ABB RobotStudio station: PickPlace_Station.rspag

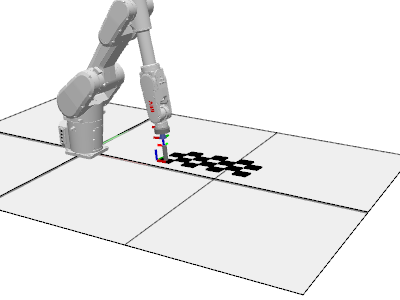
--- station ---
Station PickPlace_Station (saved by RobotStudio 24.3.10835.0)
Controller Controller1
  mechanical unit ROB_1: IRB1300F_7_140__01, 6 joints, base frame (0, 0, 0) mm
Layout (positions relative to the parent item):
  - IRB1300F_7_140__01 [mechanism, from %ABB.RobotStudio.Models.IRB1300%\IRB1300F_7_140__01.rslib] at (0, 0, 0) mm; joint values [-0.071, 0.5331, 0.806, 0.0627, 0.1234, -0.1329] (rad or m)
  - Vacuum 1x1 [part, from User Files\Vacuum 1x1.rslib] at (644.53, -45.15, 299.98) mm, rotated rx -180 ry 6.24 rz 180 deg
  - BlackSquare [part], size 100 x 60 x 10 mm
  - ChessBoard [graphiccomponentgroup] at (-2.34, 163.38, 0) mm, rotated rx 1.02 ry -6.15 rz -9.46 deg
    - MatrixRepeater [smart component, from Components\MatrixRepeater.rslib] at (653.18, -125.32, 0) mm
        properties: Source=BlackSquare; CountX=4; CountY=2; CountZ=1; OffsetX=0.2; OffsetY=0.12; OffsetZ=0.1
      - Objet_1 [part], size 100 x 60 x 10 mm
      - Objet_1 [part] at (200, 0, 0) mm, size 100 x 60 x 10 mm
      - Objet_1 [part] at (400, 0, 0) mm, size 100 x 60 x 10 mm
      - Objet_1 [part] at (600, 0, 0) mm, size 100 x 60 x 10 mm
      - Objet_1 [part] at (0, 120, 0) mm, size 100 x 60 x 10 mm
      - Objet_1 [part] at (200, 120, 0) mm, size 100 x 60 x 10 mm
      - Objet_1 [part] at (400, 120, 0) mm, size 100 x 60 x 10 mm
      - Objet_1 [part] at (600, 120, 0) mm, size 100 x 60 x 10 mm
    - MatrixRepeater_2 [smart component, from Components\MatrixRepeater.rslib] at (751.9, -66.74, 0) mm
        properties: Source=BlackSquare; CountX=3; CountY=2; CountZ=1; OffsetX=0.2; OffsetY=0.12; OffsetZ=0.1
      - Objet_1 [part], size 100 x 60 x 10 mm
      - Objet_1 [part] at (200, 0, 0) mm, size 100 x 60 x 10 mm
      - Objet_1 [part] at (400, 0, 0) mm, size 100 x 60 x 10 mm
      - Objet_1 [part] at (0, 120, 0) mm, size 100 x 60 x 10 mm
      - Objet_1 [part] at (200, 120, 0) mm, size 100 x 60 x 10 mm
      - Objet_1 [part] at (400, 120, 0) mm, size 100 x 60 x 10 mm
  - King [part] at (672.02, -45.09, 83.71) mm, rotated rx 0 ry -6.24 rz 0 deg, size 30 x 29.9 x 100 mm
Attachment: Vacuum 1x1 is attached to IRB1300F_7_140__01 / Link6
Attachment: myWobj is attached to ChessBoard
EventTableEntry 3606: ActivationMode=2, Cyclic=false, Group=, Trigger=DO_Gripper 3607, Actions=[EventTableActionAttach 3608], Comment=
EventTableTriggerIO 3607: Operator=0, IOValue=[1], IRC5Controller=? -1, SignalSource=Controller1 2384
EventTableActionAttach 3608: MountObject=false, FlangeIndext=0, FindNearest=false, AttachmentParent=Vacuum 1x1 3582, AttachmentChild=King 3605, Offset=[X=1, Y=0, Z=0, W=0, X=0, Y=1, Z=0, W=0, X=0, Y=0, Z=1, W=0, X=0, Y=0, Z=0, W=1]
EventTableTriggerIO 3609: Operator=0, IOValue=[0], IRC5Controller=? -1, SignalSource=Controller1 2384
EventTableEntry 3610: ActivationMode=2, Cyclic=false, Group=, Trigger=DO_Gripper 3609, Actions=[EventTableActionDetach 3611], Comment=
EventTableActionDetach 3611: AttachmentParent=Vacuum 1x1 3582, AttachmentChild=King 3605

--- Controller Data/Controller1/RAPID/TASK1/PROGMOD/PickPlace.modx ---
MODULE PickPlace
    CONST num nZOffset:=50;
    CONST num nGripperPickTime:=0.7;
    CONST num nGripperPlaceTime:=0.2;
    CONST num nColumnCount:=7;
    CONST num nRowCount:=4;
    CONST num nLevelCount:=1;
    CONST num nColumnSpacing:=100;
    CONST num nRowSpacing:=60;
    CONST num nLevelSpacing:=80;
    VAR errnum ERR_INDEX:=-1;
    CONST speeddata vPickPlace:=v1000;
    CONST zonedata zRefZone:=z20;

    TASK PERS tooldata myTool:=[TRUE,[[0,0,70],[1,0,0,0]],[1,[0,0,1],[1,0,0,0],0,0,0]];
    TASK PERS wobjdata myWobj:=[FALSE,TRUE,"",[[616.792188266,-66.999,77.719439522],[0.99515777,0.00445988,-0.054214569,-0.081865151]],[[0,0,0],[1,0,0,0]]];
    TASK PERS loaddata loadPart:=[0.2,[0,0,50],[1,0,0,0],0,0,0];

    ! Point 00 (Matrix Origin)
    CONST robtarget pMatrixOrigin:=[[47.449599049,30.002484299,97.931915057],[0.000000001,-0.081986553,0.996633436,-0.000000003],[-1,-1,-1,0],[9E+09,9E+09,9E+09,9E+09,9E+09,9E+09]];

    !   y
    !   ^
    !   |  +----+----+----+----+----+----+----+
    !   |  | 21 | 22 | 23 | 24 | 25 | 26 | 27 |
    !   |  +----+----+----+----+----+----+----+
    !   |  | 14 | 15 | 16 | 17 | 18 | 19 | 20 |
    !   |  +----+----+----+----+----+----+----+
    !   |  | 07 | 08 | 09 | 10 | 11 | 12 | 13 |
    !   |  +----+----+----+----+----+----+----+
    !   |  | 00 | 01 | 02 | 03 | 04 | 05 | 06 |
    !   |  +----+----+----+----+----+----+----+
    !   |
    !   +-----------------------------------> x
    !   z
    !
    PROC main()
        ! Example usage
        SetDO DO_Gripper, 0;
        PerformMatrixOperation 0,\pick;
        PerformMatrixOperation 20,\place;
        PerformMatrixOperation 20,\pick;
        PerformMatrixOperation 9,\place;
        PerformMatrixOperation 9,\pick;
        PerformMatrixOperation 4,\place;
        PerformMatrixOperation 4,\pick;
        PerformMatrixOperation 0,\place;
    ENDPROC

    PROC ControlGripper(\switch pick|switch place)
        IF Present(pick) THEN
            SetDO DO_Gripper, 1;
            GripLoad loadPart;
            WaitTime nGripperPickTime;
        ELSE
            SetDO DO_Gripper, 0;
            GripLoad load0;
            WaitTime nGripperPlaceTime;
        ENDIF
    ENDPROC

    PROC PickWithZOffset(robtarget pPick)
        VAR zonedata zonePick;
        zonePick := zRefZone;
        zonePick.pzone_tcp := nZOffset/4;
        MoveJ Offs(pPick,0,0,nZOffset),vPickPlace,zonePick,myTool\WObj:=myWobj;
        MoveL pPick,vPickPlace,fine,myTool\WObj:=myWobj;
        ControlGripper\pick;
        MoveL Offs(pPick,0,0,nZOffset),vPickPlace,zonePick,myTool\WObj:=myWobj;
    ENDPROC

    PROC PlaceWithZOffset(robtarget pPlace)
        VAR zonedata zonePlace;
        zonePlace := zRefZone;
        zonePlace.pzone_tcp := nZOffset/4;
        MoveJ Offs(pPlace,0,0,nZOffset),vPickPlace,zonePlace,myTool\WObj:=myWobj;
        MoveL pPlace,vPickPlace,fine,myTool\WObj:=myWobj;
        ControlGripper\place;
        MoveL Offs(pPlace,0,0,nZOffset),vPickPlace,zonePlace,myTool\WObj:=myWobj;
    ENDPROC

    PROC PerformMatrixOperation(num nPositionIndex,\switch pick|switch place)
        VAR num nColumnIndex;
        VAR num nRowIndex;
        VAR num nLevelIndex;
        VAR robtarget pTarget;
        VAR num errorid:=4800;
        VAR errstr my_title:="Bad Position index";
        VAR errstr str1:="The position index given is negative or superior to the matrix size";

        IF nPositionIndex<0 OR nPositionIndex>=nColumnCount*nRowCount*nLevelCount THEN
            BookErrNo ERR_INDEX;
            ErrRaise "ERR_INDEX",errorid,my_title,ERRSTR_TASK,str1,ERRSTR_CONTEXT,ERRSTR_EMPTY;
        ENDIF

        nColumnIndex:=nPositionIndex MOD nColumnCount;
        nRowIndex:=(nPositionIndex DIV nColumnCount) MOD nRowCount;
        nLevelIndex:=nPositionIndex DIV (nColumnCount*nRowCount);

        pTarget:=Offs(pMatrixOrigin,nColumnIndex*nColumnSpacing,nRowIndex*nRowSpacing,nLevelIndex*nLevelSpacing);

        IF Present(pick) THEN
            PickWithZOffset pTarget;
        ELSE
            PlaceWithZOffset pTarget;
        ENDIF
    ERROR
        IF ERRNO=ERR_INDEX THEN
            RETURN ;
        ENDIF
    ENDPROC

    FUNC bool IsPositionValid(num nPositionIndex)
        RETURN nPositionIndex>=0 AND nPositionIndex<nColumnCount*nRowCount*nLevelCount;
    ENDFUNC

    PROC syncRS()
        MoveL pMatrixOrigin,vPickPlace,fine,myTool\WObj:=myWobj;
    ENDPROC
ENDMODULE

--- Controller Data/Controller1/SYSPAR/EIO.cfg ---
EIO:CFG_1.0:7:0::
#
VIRTUAL_NETWORK:

      -Name "Virtual" -Label "Virtual Device Network"
#
EIO_SIGNAL:

      -Name "DO_Gripper" -SignalType "DO" -Access "All"

#CTRL_SIGNATURE:YWha+592Hf3kCNSwivISbM49j2HlKAlrq0MRmSSEDcIWktfFqaC8JSy5kwR+m1ZtyTd38OmdHiRdtE82Eb5awg==

--- Controller Data/Controller1/SYSPAR/PROC.cfg ---
PROC:CFG_1.0:7:0::

#CTRL_SIGNATURE:7Wf3v8outTPvk4itNNUz+JMJMk2o9zmfjYkEvuLsZsCbPvMuPL0T1QnYbu8Z0mz58Nw+3ARGvceK4pzoaQRDpA==
